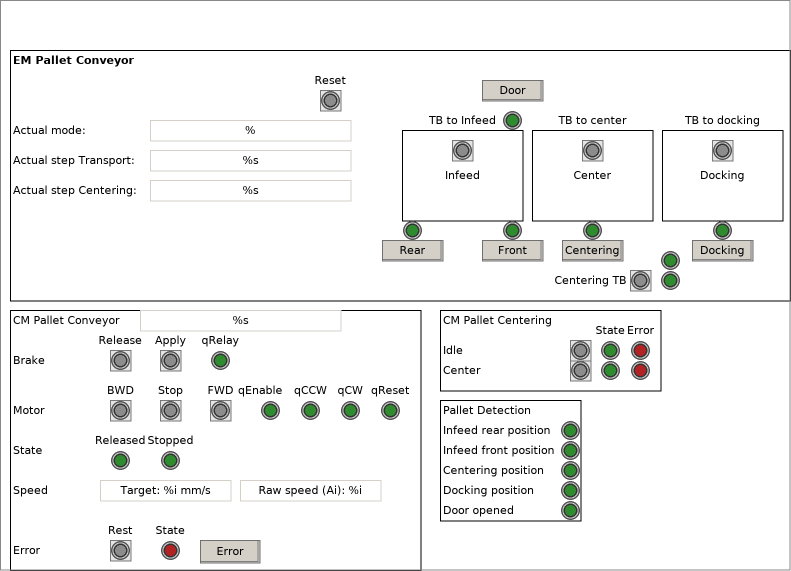
VISUALIZATION PalletConveyor_Overview  // 791x571
    Rectangle (10,50 781x251)
    Rectangle (10,310 411x261)
    Rectangle (662,130 121x91), "Docking"
    Rectangle (532,130 121x91), "Center"
    Rectangle (402,130 121x91), "Infeed"
    Label (10,50 141x21), "EM Pallet Conveyor"
    Label (550,270 81x21), "Centering TB"
    PushSwitch (630,270 21x21), variable: GVL_Modules.g_emPalletConveyor.s_fbHmiBtnTB_Centering.s_bFromHmiPressed, behaviour: TAP, style: Switch-PushSwitch-Gray
    Label (380,130 78x30)
    PushSwitch (452,140 21x21), variable: GVL_Modules.g_emPalletConveyor.s_fbHmiBtnTB_ToInfeed.s_bFromHmiPressed, behaviour: TAP, style: Switch-PushSwitch-Gray
    Label (402,110 121x21), "TB to Infeed"
    Label (532,110 121x21), "TB to center"
    Label (662,110 121x21), "TB to docking"
    PushSwitch (712,140 21x21), variable: GVL_Modules.g_emPalletConveyor.s_fbHmiBtnTB_ToDocking.s_bFromHmiPressed, behaviour: TAP, style: Switch-PushSwitch-Gray
    PushSwitch (582,140 21x21), variable: GVL_Modules.g_emPalletConveyor.s_fbHmiBtnTB_ToCentering.s_bFromHmiPressed, behaviour: TAP, style: Switch-PushSwitch-Gray
    Lamp1 (402,220 21x21), variable: GVL_Modules.g_emPalletConveyor.s_fbHmiLedInfeedRearPosition.i_bStaLed, style: Lamp-Lamp1-Green
    Lamp1 (502,220 21x21), variable: GVL_Modules.g_emPalletConveyor.s_fbHmiLedInfeedFrontPosition.i_bStaLed, style: Lamp-Lamp1-Green
    Lamp1 (582,220 21x21), variable: GVL_Modules.g_emPalletConveyor.s_fbHmiLedCenteringPosition.i_bStaLed, style: Lamp-Lamp1-Green
    Lamp1 (712,220 21x21), variable: GVL_Modules.g_emPalletConveyor.s_fbHmiLedDockingPosition.i_bStaLed, style: Lamp-Lamp1-Green
    Lamp1 (502,110 21x21), variable: GVL_Modules.g_emPalletConveyor.s_fbHmiLedDoorOpened.i_bStaLed, style: Lamp-Lamp1-Green
    Label (390,150 81x30)
    Button (382,240 61x21), "Rear"
        OnMouseClick: toggle GVL_Modules.g_emPalletConveyor.s_diStaAtInfeedPositionRear.I_bStaInput
    Button (692,240 61x21), "Docking"
        OnMouseClick: toggle GVL_Modules.g_emPalletConveyor.s_diStaAtDockingPosition.I_bStaInput
    Button (482,240 61x21), "Front"
        OnMouseClick: toggle GVL_Modules.g_emPalletConveyor.s_diStaAtInfeedPositionFront.I_bStaInput
    Button (562,240 61x21), "Centering"
        OnMouseClick: toggle GVL_Modules.g_emPalletConveyor.s_diStaAtCenteringPosition.I_bStaInput
    Button (482,80 61x21), "Door"
        OnMouseClick: toggle GVL_Modules.g_emPalletConveyor.s_diStaDoorOpened.I_bStaInput
    Button (200,540 60x23), "Error"
        OnMouseClick: toggle GVL_Modules.g_emPalletConveyor.s_cmPalletConveyor.I_bStaReadyForOperation
    Lamp1 (110,450 21x21), variable: GVL_Modules.g_emPalletConveyor.s_cmPalletConveyor.s_fbHmiLedBrakeReleased.i_bStaLed, style: Lamp-Lamp1-Green
    Lamp1 (160,540 21x21), variable: GVL_Modules.g_emPalletConveyor.s_cmPalletConveyor.s_fbHmiLedDriveError.i_bStaLed, style: Lamp-Lamp1-Red
    Textfield (240,480 141x21), "Raw speed (Ai): %i", text variable: GVL_Modules.g_emPalletConveyor.s_cmPalletConveyor.Q_nSetTargetSpeed
    Textfield (100,480 131x21), "Target: %i mm/s", text variable: GVL_Modules.g_emPalletConveyor.s_cmPalletConveyor.s_fTargetSpeed, input disabled if: 0
        OnMouseClick: write the text variable via VisuDialogs.Numpad, min 40, max 200
    Lamp1 (300,400 21x21), variable: GVL_Modules.g_emPalletConveyor.s_cmPalletConveyor.Q_bCmdStartCCW, style: Lamp-Lamp1-Green
    Lamp1 (210,350 21x21), variable: GVL_Modules.g_emPalletConveyor.s_cmPalletConveyor.Q_bCmdReleaseBrake, style: Lamp-Lamp1-Green
    Lamp1 (340,400 21x21), variable: GVL_Modules.g_emPalletConveyor.s_cmPalletConveyor.Q_bCmdStartCW, style: Lamp-Lamp1-Green
    Label (10,310 131x21), "CM Pallet Conveyor"
    PushSwitch (160,350 21x21), variable: GVL_Modules.g_emPalletConveyor.s_cmPalletConveyor.s_fbHmiBtnManualApplyBrake.s_bFromHmiPressed, behaviour: TAP, style: Switch-PushSwitch-Gray
    PushSwitch (110,350 21x21), variable: GVL_Modules.g_emPalletConveyor.s_cmPalletConveyor.s_fbHmiBtnManualReleaseBrake.s_bFromHmiPressed, behaviour: TAP, style: Switch-PushSwitch-Gray
    Label (140,330 61x21), "Apply"
    Label (190,330 61x21), "qRelay"
    Label (90,430 61x21), "Released"
    Label (90,330 61x21), "Release"
    Label (10,350 101x21), "Brake"
    Label (10,400 101x21), "Motor"
    Lamp1 (160,450 21x21), variable: GVL_Modules.g_emPalletConveyor.s_cmPalletConveyor.s_fbHmiLedMotorStopped.i_bStaLed, style: Lamp-Lamp1-Green
    PushSwitch (110,400 21x21), variable: GVL_Modules.g_emPalletConveyor.s_cmPalletConveyor.s_fbHmiBtnManualBackward.s_bFromHmiPressed, behaviour: TAP, style: Switch-PushSwitch-Gray
    PushSwitch (160,400 21x21), variable: GVL_Modules.g_emPalletConveyor.s_cmPalletConveyor.s_fbHmiBtnManualStop.s_bFromHmiPressed, behaviour: TAP, style: Switch-PushSwitch-Gray
    PushSwitch (210,400 21x21), variable: GVL_Modules.g_emPalletConveyor.s_cmPalletConveyor.s_fbHmiBtnManualForward.s_bFromHmiPressed, behaviour: TAP, style: Switch-PushSwitch-Gray
    Label (90,380 61x21), "BWD"
    Label (140,380 61x21), "Stop"
    Label (190,380 61x21), "FWD"
    Label (140,430 61x21), "Stopped"
    Label (10,540 101x21), "Error"
    Label (140,520 61x21), "State"
    PushSwitch (110,540 21x21), variable: GVL_Modules.g_emPalletConveyor.s_cmPalletConveyor.s_fbHmiBtnManualReset.s_bFromHmiPressed, behaviour: TAP, style: Switch-PushSwitch-Gray
    Label (90,520 61x21), "Rest"
    Label (280,380 61x21), "qCCW"
    Label (320,380 61x21), "qCW"
    Label (10,480 101x21), "Speed"
    Rectangle (440,400 141x121)
    Lamp1 (560,420 21x21), variable: GVL_Modules.g_emPalletConveyor.s_fbHmiLedInfeedRearPosition.i_bStaLed, style: Lamp-Lamp1-Green
    Label (440,420 121x21), "Infeed rear position"
    Label (455,486 78x30)
    Label (440,400 121x21), "Pallet Detection"
    Lamp1 (560,440 21x21), variable: GVL_Modules.g_emPalletConveyor.s_fbHmiLedInfeedFrontPosition.i_bStaLed, style: Lamp-Lamp1-Green
    Lamp1 (560,460 21x21), variable: GVL_Modules.g_emPalletConveyor.s_fbHmiLedCenteringPosition.i_bStaLed, style: Lamp-Lamp1-Green
    Lamp1 (560,480 21x21), variable: GVL_Modules.g_emPalletConveyor.s_fbHmiLedDockingPosition.i_bStaLed, style: Lamp-Lamp1-Green
    Lamp1 (560,500 21x21), variable: GVL_Modules.g_emPalletConveyor.s_fbHmiLedDoorOpened.i_bStaLed, style: Lamp-Lamp1-Green
    Label (440,440 121x21), "Infeed front position"
    Label (440,460 121x21), "Centering position"
    Label (440,480 121x21), "Docking position"
    Label (440,500 121x21), "Door opened"
    Rectangle (440,310 221x81)
    Lamp1 (600,340 21x21), variable: GVL_Modules.g_emPalletConveyor.s_cmCenteringUnit.s_fbHmiLedIsOff.i_bStaLed, style: Lamp-Lamp1-Green
    Lamp1 (630,340 21x21), variable: GVL_Modules.g_emPalletConveyor.s_cmCenteringUnit.s_fbHmiLedErrorOff.i_bStaLed, style: Lamp-Lamp1-Red
    PushSwitch (570,360 21x21), variable: GVL_Modules.g_emPalletConveyor.s_cmCenteringUnit.s_fbHmiBtnManualOn.s_bFromHmiPressed, behaviour: TAP, style: Switch-PushSwitch-Gray
    PushSwitch (570,340 21x21), variable: GVL_Modules.g_emPalletConveyor.s_cmCenteringUnit.s_fbHmiBtnManualOff.s_bFromHmiPressed, behaviour: TAP, style: Switch-PushSwitch-Gray
    Label (440,340 91x21), "Idle"
    Label (440,360 78x21), "Center"
    Label (440,310 141x21), "CM Pallet Centering"
    Lamp1 (600,360 21x21), variable: GVL_Modules.g_emPalletConveyor.s_cmCenteringUnit.s_fbHmiLedIsOn.i_bStaLed, style: Lamp-Lamp1-Green
    Lamp1 (630,360 21x21), variable: GVL_Modules.g_emPalletConveyor.s_cmCenteringUnit.s_fbHmiLedErrorOn.i_bStaLed, style: Lamp-Lamp1-Red
    Label (590,320 41x21), "State"
    Label (620,320 41x21), "Error"
    Label (10,150 131x21), "Actual step Transport:"
    PushSwitch (320,90 21x21), variable: GVL.g_unCleanroomConnect.s_fbHmiBtnReset.s_bFromHmiPressed, behaviour: TAP, style: Switch-PushSwitch-Gray
    Textfield (150,150 201x21), "%s", text variable: GVL_Modules.g_emPalletConveyor.s_fbSeqTransportControl.i_sStepName
    Label (310,70 41x21), "Reset"
    Label (10,120 131x21), "Actual mode:"
    Label (10,180 131x21), "Actual step Centering:"
    Textfield (150,180 201x21), "%s", text variable: GVL_Modules.g_emPalletConveyor.s_fbSeqCenteringControl.i_sStepName
    Textfield (150,120 201x21), "%", text list: 'E_MODE', text index: GVL_Modules.g_emPalletConveyor.i_eCtrlMode
    Textfield (140,310 201x21), "%s", text variable: GVL_Modules.g_emPalletConveyor.s_cmPalletConveyor.s_sActStep
    Lamp1 (380,400 21x21), variable: GVL_Modules.g_emPalletConveyor.s_cmPalletConveyor.Q_bCmdReset, style: Lamp-Lamp1-Green
    Label (360,380 61x21), "qReset"
    Lamp1 (260,400 21x21), variable: GVL_Modules.g_emPalletConveyor.s_cmPalletConveyor.Q_bCmdEnable, style: Lamp-Lamp1-Green
    Label (230,380 61x21), "qEnable"
    Label (10,440 101x21), "State"
    Lamp1 (660,250 21x21), variable: GVL_Modules.g_emPalletConveyor.s_fbHmiLedCenteringCenter.i_bStaLed, style: Lamp-Lamp1-Green
    Lamp1 (660,270 21x21), variable: GVL_Modules.g_emPalletConveyor.s_fbHmiLedCenteringIdle.i_bStaLed, style: Lamp-Lamp1-Green
END_VISUALIZATION

(* stored: Version 1.1.0.1, ProductVersion 3.1.4024.12
   Visu PalletConveyor_Overview: Id {7e703562-77b6-483e-8a23-ae70d8327860} *)
